// TIA Portal V20 export
TYPE "MABS_ManIn"
// stored: Access Published, Namespace LineB1
   STRUCT
      RunBalls : Bool;
      Switch : Struct
         ToLeft : Bool;
         ToRight : Bool;
         left_to_st : Bool;
         right_to_st : Bool;
      END_STRUCT;
   END_STRUCT;
END_TYPE
